{attribute 'GeneratedUsingTerminal: EJ1957-0000-0017'}
{attribute addProperty BoxType "EJ1957-0000-0017"}
{attribute addProperty Id "OutputsOutputs_7EDA7A424"}
{attribute addProperty CRC "1515908004"}
{attribute addProperty Size "4"}
TYPE Module_2_FSOUT_5A5AEBA4 :
STRUCT
	{attribute addProperty Name "Outputs"}
	Outputs  : Outputs_7EDA7A42;
END_STRUCT
END_TYPE

(* stored: Version 1.2.0.0, ProductVersion 3.1.4024.11
   DUT Module_2_FSOUT_5A5AEBA4: Id {0b71c5f5-f9df-4217-8d9e-a9468844b67d} *)
